Staubli VAL3: JPOINT.pjx

--- JPOINT.pjx ---
Parameters version=s7.6.1 stackSize=5000 millimeterUnit=true
Program file=computeFrame.pgx
Program file=delete.pgx
Program file=deleteItem.pgx
Program file=duplicate.pgx
Program file=find.pgx
Program file=get.pgx
Program file=getDistance.pgx
Program file=getFrame.pgx
Program file=getFrameId.pgx
Program file=getFunctionEdit.pgx
Program file=getFunctionSel.pgx
Program file=getFunctionView.pgx
Program file=getListItem.pgx
Program file=getPoint.pgx
Program file=getSize.pgx
Program file=getSizeItem.pgx
Program file=getTool.pgx
Program file=getTrajItem.pgx
Program file=getTrajType.pgx
Program file=goTo.pgx
Program file=HerePoint.pgx
Program file=insertItem.pgx
Program file=load.pgx
Program file=loadCycle.pgx
Program file=loadPage.pgx
Program file=makeTraj.pgx
Program file=moveTo.pgx
Program file=new.pgx
Program file=onEdit.pgx
Program file=onEditItem.pgx
Program file=onFunctionEdit.pgx
Program file=onFunctionSel.pgx
Program file=onFunctionView.pgx
Program file=onInsert.pgx
Program file=onProgEnd.pgx
Program file=onRun.pgx
Program file=onSave.pgx
Program file=onStart.pgx
Program file=onStop.pgx
Program file=setFrameId.pgx
Program file=setTool.pgx
Program file=setTrajItem.pgx
Data file=JPOINT.dtx
Library alias=saveData path=Disk://saveData/saveData.pjx
Library alias=page path=Disk://kernel/template/page/page.pjx
Library alias=use path=Disk://kernel/userPage/userPage.pjx
Library alias=language path=Disk://kernel/language/language.pjx
Library alias=tcp path=Disk://kernel/tool/tool.pjx
Library alias=cycleStatus path=Disk://cycleStatus/cycleStatus.pjx
Library alias=pt path=Disk://kernel/template/session/saveTraj/JPOINT/JPOINT.pjx
Library alias=home path=Disk://kernel/template/session/saveTraj/HOME/HOME.pjx
Type name=TrajectoryItem path=Disk://kernel/template/TrajectoryItem/TrajectoryItem.pjx
Type name=TrajJoint path=Disk://kernel/template/TrajJoint/TrajJoint.pjx
Type name=ActionItem path=Disk://kernel/template/ActionItem/ActionItem.pjx
Type name=InstrItem path=Disk://kernel/template/InstrItem/InstrItem.pjx
Type name=Trajectory path=Disk://kernel/template/Trajectory/Trajectory.pjx
Type name=TrajHome path=Disk://kernel/template/TrajHome/TrajHome.pjx
Type name=FrameItem path=Disk://kernel/template/FrameItem/FrameItem.pjx

--- JPOINT.dtx ---
public string sItems
string sPathTemplate = "Disk://kernel/template/JPOINT"
public bool bMoveType[3]
public bool bStepping
pointRx pToGo = {fatherId=world[0]}
pointRx pLastPoint = {fatherId=world[0]}
mdesc nom_speed = {accel=50, vel=50, decel=50, blend=off}
num nTcpAction
pointRx pPointTo = {fatherId=world[0]}
string sTrajType
string sMenu[8]
mdesc mMdesc = {accel=25, vel=25, decel=25, blend=off}
bool bToSave
InstrItem tcpInstr
  [0]
    string sType
    string sData
public Trajectory tTraj
  [0]
    TrajectoryItem tSuper
      [0]
        num distance
        num moveType
        num nTime
        num nStop
        num nTcpAction
        string comment
        bool toStop
        mdesc nom_speed = {tmax=300, rmax=9999, leave=30, reach=30}
        InstrItem iInstr[3]
          [0]
            string sType
            string sData
          [1]
            string sType
            string sData
          [2]
            string sType
            string sData
        num nMoveId
    string sID
    num nId
num nIndex
num nKey
TrajJoint jEditPoint
  [0]
    num nIndexTool
    TrajJointItem tData
      [0]
        jointRx jJoint
        TrajectoryItem tSuper
          [0]
            num distance
            num moveType
            num nTime
            num nStop
            num nTcpAction
            string comment
            bool toStop
            mdesc nom_speed = {tmax=9999, rmax=9999, leave=30, reach=30}
            InstrItem iInstr[3]
              [0]
                string sType
                string sData
              [1]
                string sType
                string sData
              [2]
                string sType
                string sData
            num nMoveId
    string sID
    num nIndexFrame
string sTrajCycle

--- delete.pgx ---
public program delete(string x_sName, num& x_nResult[])
  local string l_sItem
  local num l_nSize
begin
  //
  // delete the select trajectory
  //
  if isDefined(pt:tTraj[x_sName])
    // delete
    delete(pt:tTraj[x_sName])
    // save it
    bToSave=true
    x_nResult=0
  else
    x_nResult=-1
  endIf

end

--- deleteItem.pgx ---
public program deleteItem(num& x_nIndex)
  local num i
  local string l_sItem
begin
  // delete the selected item
  delete(jEditPoint.tData[x_nIndex])
end

--- duplicate.pgx ---
public program duplicate(string x_sCopy, string x_sPaste, num& x_nResult[])
  local num i
  local num l_nSize
  local string l_sItem
  local bool l_bFound
  local num l_nResult
  local string l_sString
  local num l_nX
  local num l_nY
begin
  // duplicate

  // look if the items exist
  if insert(pt:tTraj[x_sPaste])
    // link the point
    call pt:copy_it(x_sCopy,x_sPaste)
    call pt:link_it(x_sPaste)
    // save it
    bToSave=true
  endIf
end

--- find.pgx ---
public program find(string& x_sItem[], bool& x_bFound[])
begin
  // check if the item has been found
  x_bFound=isDefined(pt:tTraj[x_sItem])
end

--- getDistance.pgx ---
public program getDistance(tool x_tTool, num& x_nDistance[], bool x_bCycle, num x_nIndex)
  local num l_nDistance
  local point l_pPoint
  local num l_nValue
  local trsf l_trsfEmpty
begin
  // first point
  if x_nIndex==0
    x_nDistance=10
    return
  elseIf x_bCycle
    // an other one
    x_nDistance=distance(jointToPoint(x_tTool,world,pt:tTraj[sTrajCycle].tData[x_nIndex-1].jJoint),jointToPoint(x_tTool,world,pt:tTraj[sTrajCycle].tData[x_nIndex].jJoint))
  else
     x_nDistance=distance(jointToPoint(x_tTool,world,jEditPoint.tData[x_nIndex-1].jJoint),jointToPoint(x_tTool,world,jEditPoint.tData[x_nIndex].jJoint))
  endIf
end

--- getFunctionEdit.pgx ---
public program getFunctionEdit(string& x_sName[])
  local string l_sMessage
begin
  //
  // define your message for the
  // function KEY
  //
  // NOTE is an ARRAY[0..7]
  //
  // example:
  // x_sName[1]="DEMO"
  // active the F2 button
  //
  // here
  call language:message(l_sMessage,150)
  x_sName[0]=l_sMessage
  // ALIGN
  call language:message(l_sMessage,134)
  x_sName[1]=l_sMessage
  // Tool
  call language:message(l_sMessage,123)
  x_sName[2]=l_sMessage
end

--- getFunctionSel.pgx ---
public program getFunctionSel(string& x_sName[])
  local string l_sMessage
begin
  //
  // define your message for the
  // function KEY
  //
  // NOTE is an ARRAY[0..7]
  //
  // example:
  // x_sName[1]="DEMO"
  // active the F2 button
  //
end

--- getFunctionView.pgx ---
public program getFunctionView(string& x_sName[])
  local string l_sMessage
begin
  //
  // define your message for the
  // function KEY
  //
  // NOTE is an ARRAY[0..7]
  //
  // example:
  // x_sName[1]="DEMO"
  // active the F2 button
  //
  // here
  call language:message(l_sMessage,150)
  x_sName[0]=l_sMessage
  // ALIGN
  call language:message(l_sMessage,134)
  x_sName[1]=l_sMessage
end

--- getListItem.pgx ---
public program getListItem(string& x_sItem[], num x_nIndex)
  local trsf l_tTrsf
  local string l_sItem[6]
  local string l_sEvent
begin
  //
  //
  // define the item to show in the edit page Traj
  // customize an array and copy to x_sItem...
  //
  // see other traj as example
  l_sItem[0]=("Joint 1 > "+toString(".2",jEditPoint.tData[x_nIndex].jJoint.j1))
  l_sItem[1]=("Joint 2 > "+toString(".2",jEditPoint.tData[x_nIndex].jJoint.j2))
  l_sItem[2]=("Joint 3 > "+toString(".2",jEditPoint.tData[x_nIndex].jJoint.j3))
  l_sItem[3]=("Joint 4 > "+toString(".2",jEditPoint.tData[x_nIndex].jJoint.j4))
  l_sItem[4]=("Joint 5 > "+toString(".2",jEditPoint.tData[x_nIndex].jJoint.j5))
  l_sItem[5]=("Joint 6 > "+toString(".2",jEditPoint.tData[x_nIndex].jJoint.j6))
  call use:stringCopy(l_sItem,x_sItem)
end

--- getPoint.pgx ---
public program getPoint(point& x_pPoint[], bool x_bCycle, num x_nIndex)
  local string l_sItem
  local tool l_tTool
begin
  // take
  // check the point
  link(x_pPoint,world)
  if x_bCycle
    call tcp:getTool(l_tTool,pt:tTraj[sTrajCycle].nIndexTool)
    x_pPoint=jointToPoint(l_tTool,world,pt:tTraj[sTrajCycle].tData[x_nIndex].jJoint)
  else
    // give back the point
    call tcp:getTool(l_tTool,jEditPoint.nIndexTool)
    x_pPoint=jointToPoint(l_tTool,world,jEditPoint.tData[x_nIndex].jJoint)
  endIf
end

--- getSize.pgx ---
public program getSize(num& x_nSize[])
  local string l_sType
  local string l_sKey
  local num i
  local string l_sItem
  local string l_sPath
begin
  // give back the size to trajectory field
  x_nSize=size(pt:tTraj)
end

--- getSizeItem.pgx ---
public program getSizeItem(bool x_bCycle, num& x_nSize)
  local string l_sType
  local string l_sKey
  local num i
begin
  //
  // get the size of the collection
  //
  if x_bCycle
    x_nSize=size(pt:tTraj[sTrajCycle].tData)
  else
    x_nSize=size(jEditPoint.tData)
  endIf
end

--- getTrajItem.pgx ---
public program getTrajItem(TrajectoryItem& x_tTraj[], num x_nIndex)
begin
  //
  // get all the FIELD
  //
  x_tTraj=jEditPoint.tData[x_nIndex].tSuper
end

--- goTo.pgx ---
public program goTo(tool x_tTool, mdesc x_mDesc, num x_nMoveType, bool& x_bUnreached[], num x_nIndex)
  local point l_pTrsf
  local bool l_bInside
  local tool l_tTool
  local point l_pHere
  local string l_sMessage
  local num l_nSize
  local num i
begin
  // the maximum size
  if isInRange(jEditPoint.tData[x_nIndex].jJoint)
    // go to the select Joint
    movej(jEditPoint.tData[x_nIndex].jJoint,x_tTool,x_mDesc)
  else
    x_bUnreached=true
  endIf
end

--- HerePoint.pgx ---
public program HerePoint(num x_nIndex)
  local tool l_tTool
  local point l_pHere
  local frame l_fFrame
  local num i
  local num l_nIndex
begin
  //
  // take the point
  //
  jEditPoint.tData[x_nIndex].jJoint=herej()
  resetMotion()
end

--- insertItem.pgx ---
public program insertItem(num x_nIndexCopy, num x_nIndexPaste)
  local num l_nLastType
  local point l_pPoint
  local num l_nType
  local joint l_jJoint
begin
  //
  // use to add more elements from the typical one
  //
  // insert all the field
  //
  // JOINT
  l_jJoint=jEditPoint.tData[x_nIndexCopy].jJoint
  insert(jEditPoint.tData[x_nIndexPaste])
  jEditPoint.tData[x_nIndexPaste].jJoint=l_jJoint

end

--- load.pgx ---
public program load(string x_sItem, num& x_nResult)
  local string l_sType
  local string l_sMessage
begin
  // load the select trajectory..already loaded
  call getTrajType(l_sType)
  if find(pt:libPath(),saveData:sPathTraj)==-1
    pt:libLoad(saveData:sPathTraj+l_sType)
    delay(0)
    if saveData:bDebug
      ? "loading JPOINT..."+saveData:sPathTraj+l_sType
    endIf
  endIf
  // use the type...
  if isDefined(pt:tTraj[x_sItem])
    // use the type...
    jEditPoint=pt:tTraj[x_sItem]
    jEditPoint.sID=x_sItem
    x_nResult=0
  elseIf x_sItem!="" and find(x_sItem,"@")==-1
    // not FOUND
    call language:message(l_sMessage,-7)
    x_nResult=-1
    popUpMsg(l_sMessage+x_sItem)
    jEditPoint.sID=""
  elseIf x_sItem==""
    // reload all the template
    x_nResult=home:libLoad(saveData:sPathTraj+"HOME")
    if saveData:bDebug
      ? "loading JPOINT HOME..."+saveData:sPathTraj+"HOME"
    endIf
  endIf
end

--- loadCycle.pgx ---
public program loadCycle(string x_sItem, num& x_nResult[])
  local string l_sType
  local string l_sMessage
begin
  // load the select trajectory..already loaded
  call getTrajType(l_sType)
  if find(pt:libPath(),saveData:sPathTraj)==-1
    pt:libLoad(saveData:sPathTraj+l_sType)
    delay(0)
    if saveData:bDebug
      ? "loading JPOINT..."+saveData:sPathTraj+l_sType
    endIf
  endIf
  if isDefined(pt:tTraj[x_sItem])
    // use the type...
    sTrajCycle=x_sItem
  else
    // not FOUND
    call language:message(l_sMessage,-7)
    x_nResult=-1
    cycleStatus:bToStop=true
    popUpMsg(l_sMessage+x_sItem)
  endIf
end

--- loadPage.pgx ---
program loadPage(string x_sPage, string& x_sItems[])
// load the next page
  local num i
begin
  // look if the page libload is correct
  i=page:libLoad(x_sPage)
    delay(0)
  logMsg("KERNEL:PAGE LIBLOAD "+x_sPage+" result "+toString("",i))
  if i!=0
    popUpMsg("Loading page "+x_sPage+" error CODE "+toString("",i))
  else
    page:sItems=x_sItems
    call page:main()
  endIf
end

--- makeTraj.pgx ---
public program makeTraj(string& x_sItem[])
  local num i
  local num l_nSize
  local tool l_tTool
  local bool l_bUnreached
  local point l_pPoint[2]
  local num l_nMoveId
  local bool l_bOk
  local ActionItem l_aAction
  local num j
  local TrajectoryItem l_tTraj
  local num l_nDistance
  local joint l_jJoint
  local Trajectory l_tTrajectory
begin
  //
  // inizialize the system
  //
  // take the TOOL
  call tcp:getTool(l_tTool,pt:tTraj[sTrajCycle].nIndexTool)
  //
  // for all of my traj cycleJoint move the robot
  //
  // the maximum size
  call getSizeItem(true,l_nSize)
  //
  // for all of my traj cyclePoints move the robot
  //
  resize(tTraj.tSuper,1,size(pt:tTraj[sTrajCycle].tData))
  for i=0 to (l_nSize-1)
    tTraj.tSuper[i]=pt:tTraj[sTrajCycle].tData[i].tSuper
  endFor
  tTraj.sID="JPOINT "+pt:tTraj[sTrajCycle].sID
  call cycleStatus:addTraj(tTraj)
  for i=0 to (l_nSize-1)
    //
    // get the point info
    //
    l_tTraj=pt:tTraj[sTrajCycle].tData[i].tSuper
    //
    // get the distance in percentage
    //
    call getDistance(l_tTool,l_nDistance,true,i)
    //
    // give to the traj library the percentage distance
    //
    if l_tTraj.toStop
      l_tTraj.nom_speed.blend=off
    endIf
    //
    // put the move in the stack
    //
    l_jJoint=pt:tTraj[sTrajCycle].tData[i].jJoint
    call moveTo(l_tTool,l_tTraj.nom_speed,l_tTraj.moveType,l_bUnreached,l_jJoint,l_nMoveId)
    // set the data
    l_aAction.nDistance=l_nDistance
    l_aAction.nPointId=i
    l_aAction.nMoveId=l_nMoveId
    l_aAction.sIdTraj="JPOINT "+pt:tTraj[sTrajCycle].sID
    call cycleStatus:putInstr_Traj(l_aAction,l_tTraj,pt:tTraj[sTrajCycle].nIndexTool,l_nSize)
    // there is a waitEndMove
    if l_tTraj.toStop
      waitEndMove()
      delay(l_tTraj.nStop)
      // wait all the action has been done
      wait(cycleStatus:bActionRunning==false)
    endIf
  endFor
end

--- moveTo.pgx ---
public program moveTo(tool x_tTool, mdesc x_mDesc, num x_nMoveType, bool& x_bUnreached[], joint& x_jJoint[], num& x_nMoveId)
begin
  //
  // use the percentage speed
  //
  x_mDesc.vel=saveData:nSpeed/100*x_mDesc.vel
  x_nMoveId=movej(x_jJoint,x_tTool,x_mDesc)
end

--- onEdit.pgx ---
public program onEdit(string& x_sItem[])
  local string l_sPath
  local num i
  local string l_sItem
  local num l_nSize
  local TrajectoryItem l_tTraj
  local num l_nResult
  local string l_sPoint
begin
  // DEFINE YOUR ITEM
  call getTrajType(saveData:sTrajTypeUsing)
  // load the trajectory
  call load(x_sItem,l_nResult)
  if find(x_sItem,"@")==-1
    // load the page viewTraj
    l_sPath="Disk://trajectory/page_viewTraj"
    // give back the path
    x_sItem[1]=x_sItem
    x_sItem=l_sPath
  endIf
end

--- onEditItem.pgx ---
public program onEditItem(string& x_sEvent[], num x_nIndex, num x_nIndexItem)
  local joint l_jJoint
  local num i
  local string l_sEmpty
  local string l_sMessage
begin
  // edit the custom element that was add in the list
  l_jJoint=jEditPoint.tData[x_nIndexItem].jJoint
  call use:findPos(x_sEvent,">",i)
  i=i+1
  // clean the line
  call use:listcursor(use:nView,false)
  l_sEmpty=""
  switch x_nIndex
    case 0
      //  j1-value
      if cycleStatus:bCycle
        // set a limit +- 5
        call use:changeValue(l_jJoint.j1,l_jJoint.j1-5,l_jJoint.j1+5,i+40-use:nBottomX,use:nView+1,l_sEmpty)
      else
        call use:changeValue(l_jJoint.j1,0,0,i+40-use:nBottomX,use:nView+1,l_sEmpty)
      endIf
    break
    case 1
      //  j2-value
      if cycleStatus:bCycle
        // set a limit +- 5
        call use:changeValue(l_jJoint.j2,l_jJoint.j2-5,l_jJoint.j2+5,i+40-use:nBottomX,use:nView+1,l_sEmpty)
      else
        call use:changeValue(l_jJoint.j2,0,0,i+40-use:nBottomX,use:nView+1,l_sEmpty)
      endIf
    break
    case 2
      //  j3-value
      if cycleStatus:bCycle
        // set a limit +- 5
        call use:changeValue(l_jJoint.j3,l_jJoint.j3-5,l_jJoint.j3+5,i+40-use:nBottomX,use:nView+1,l_sEmpty)
      else
        call use:changeValue(l_jJoint.j3,0,0,i+40-use:nBottomX,use:nView+1,l_sEmpty)
      endIf
    break
    case 3
      //  j4-value
      if cycleStatus:bCycle
        // set a limit +- 5
        call use:changeValue(l_jJoint.j4,l_jJoint.j4-5,l_jJoint.j4+5,i+40-use:nBottomX,use:nView+1,l_sEmpty)
      else
        call use:changeValue(l_jJoint.j4,0,0,i+40-use:nBottomX,use:nView+1,l_sEmpty)
      endIf
    break
    case 4
      //  j5-value
      if cycleStatus:bCycle
        // set a limit +- 5
        call use:changeValue(l_jJoint.j5,l_jJoint.j5-5,l_jJoint.j5+5,i+40-use:nBottomX,use:nView+1,l_sEmpty)
      else
        call use:changeValue(l_jJoint.j5,0,0,i+40-use:nBottomX,use:nView+1,l_sEmpty)
      endIf
    break
    case 5
      //  j6-value
      if cycleStatus:bCycle
        // set a limit +- 5
        call use:changeValue(l_jJoint.j6,l_jJoint.j6-5,l_jJoint.j6+5,i+40-use:nBottomX,use:nView+1,l_sEmpty)
      else
        call use:changeValue(l_jJoint.j6,0,0,i+40-use:nBottomX,use:nView+1,l_sEmpty)
      endIf
    break
  endSwitch
  //
  if isInRange(l_jJoint)
    jEditPoint.tData[x_nIndexItem].jJoint=l_jJoint
  else
    // error using the trsf
    call language:message(l_sMessage,-5)
    popUpMsg(l_sMessage)
  endIf
  // wait no key
  call use:nullKey(nKey)
end

--- onFunctionEdit.pgx ---
public program onFunctionEdit(num x_nIndex, string x_sEvent, num x_nFunctionKey)
  local string l_sMessage
  local string l_sButton[2]
  local bool l_bOk
  local string l_sPage
  local string l_sItem
  local tool l_tTool
  local point l_pAlign
  local bool l_bYes
  local string l_sMessage2
begin
  //
  // do on Key action
  //
  // x_nIndex = actual index item
  // x_sEvent = actual event item
  //
  switch x_nFunctionKey
    // F1 button
    case 271
      // HERE JOINT
      if !cycleStatus:bCycle
        call language:message(l_sMessage,160)
        call language:getYesNo(l_sButton)
        // ask the yes_no question
        call use:yes_no(l_sMessage,l_sButton,l_bYes)
        if l_bYes
          call HerePoint(x_nIndex)
        endIf
      endIf
    break
    case 272
      // ALIGN
      if !cycleStatus:bCycle
        resetMotion()
        // tool
        call tcp:getTool(l_tTool,jEditPoint.nIndexTool)
        l_pAlign=here(l_tTool,world)
        l_pAlign.trsf=align(l_pAlign.trsf,saveData:fFrameItem[saveData:nFrameActive].fFrame.trsf)
        call language:message(l_sMessage,203)
        call language:message(l_sMessage2,134)
        l_sMessage=l_sMessage+" "+l_sMessage2+"..."
        call use:timerDialog(l_sMessage,0)
        movej(l_pAlign,l_tTool,mMdesc)
        watch(isEmpty() or isKeyPressed(255),3)
        if !isEmpty()
          resetMotion()
        endIf
        delay(2)
      endIf
    break
    // F3 button
    case 273
      // Select the gun
      l_sPage="Disk://kernel/page/tool"
      call loadPage(l_sPage,l_sItem)
      // set the tool
      jEditPoint.nIndexTool=saveData:nIndexTool
    break
    // F4 button
    case 274
    break
    // F5 button
    case 275
    break
    // F6 button
    case 276
    break
    // F7 button
    case 277
    break
    // F8 button
    case 278
      // save it
    break
  endSwitch
end

--- onFunctionSel.pgx ---
public program onFunctionSel(num x_nIndex, string& x_sEvent, num x_nFunctionKey)
  local num l_nX
  local num l_nY
  local string l_sString
  local string l_sName
begin
  //
  // do on Key action
  //
  // x_nIndex = actual index item
  // x_sEvent = actual event item
  //
  l_nX=40-use:nBottomX-1
  l_nY=use:nBottomY+1
  switch x_nFunctionKey
    // F1 button
    case 271
    break
    // F2 button
    case 272
    break
    // F3 button
    case 273
    break
    // F4 button
    case 274
    break
    // F5 button
    case 275
    break
    // F6 button
    case 276
    break
    // F7 button
    case 277
    break
    // F8 button
    case 278
      //      call language:message(l_sString,21)
      //      call use:type(l_nX,l_nY,l_sString)
      //      // read the new trajectory
      //      call use:read(l_nX+len(l_sString),l_nY,l_sName,10,false)
      //      if !use:bUseEscape
      //        // look if the items exist
      //        if insert(pt:tTraj[l_sName])
      //          call pt:link_it(l_sName)
      //          pt:tTraj[l_sName].nIndexTool=saveData:nIndexTool
      //          // save it
      //          bToSave=true
      //          // export
      //          x_sEvent=l_sName
      //        else
      //          call language:message(l_sString,-2)
      //          popUpMsg(l_sString)
      //        endIf
      //      endIf
    break
  endSwitch
end

--- onFunctionView.pgx ---
public program onFunctionView(num x_nIndex, string x_sEvent, num x_nFunctionKey)
  local string l_sMessage
  local string l_sButton[2]
  local bool l_bYes
  local tool l_tTool
  local point l_pAlign
  local string l_sMessage2
  local joint l_jJoint
  local num l_nIndexFrame
  local frame l_fFrame
begin
  //
  // do on Key action
  //
  // x_nIndex = actual index item
  // x_sEvent = actual event item
  //
  switch x_nFunctionKey
    // F1 button
    case 271
      // HERE JOINT
      if !cycleStatus:bCycle
        call language:message(l_sMessage,160)
        call language:getYesNo(l_sButton)
        // ask the yes_no question
        call use:yes_no(l_sMessage,l_sButton,l_bYes)
        if l_bYes
          call HerePoint(x_nIndex)
        endIf
      endIf
    break
    // F2 button
    case 272
      // ALIGN
      if !cycleStatus:bCycle and !cycleStatus:bSimulation
        resetMotion()
        call getFrameId(l_nIndexFrame)
        l_fFrame=saveData:fFrameItem[l_nIndexFrame].fFrame
        // tool
        call tcp:getTool(l_tTool,jEditPoint.nIndexTool)
        l_pAlign=here(l_tTool,l_fFrame)
        l_pAlign.trsf=align(l_pAlign.trsf,l_fFrame.trsf)
        // check the align
        if pointToJoint(l_tTool,herej(),l_pAlign,l_jJoint)
          call language:message(l_sMessage,203)
          call language:message(l_sMessage2,134)
          l_sMessage=l_sMessage+" "+l_sMessage2+"..."
          call use:timerDialog(l_sMessage,0)
          movel(l_pAlign,l_tTool,mMdesc)
          watch(isEmpty() or isKeyPressed(255),3)
          if !isEmpty()
            resetMotion()
          endIf
          delay(2)
        endIf
      endIf
    break
    // F3 button
    case 273
    break
    // F4 button
    case 274
    break
    // F5 button
    case 275
    break
    // F6 button
    case 276
    break
    // F7 button
    case 277
    break
    // F8 button
    case 278
    break
  endSwitch
end

--- onInsert.pgx ---
public program onInsert(string& x_sItem[])
  local string l_sEvent
  local num l_nKey
  local num l_nIndex
  local num l_nSize
  local num i
  local string l_sMessage
  local bool l_bFound
  local string l_sType
  local bool l_bUseFilter
  local string l_sPaste
  local num l_nResult
  local num l_nX
  local num l_nY
  local string l_sName
begin
  // get the type
  call getTrajType(x_sItem)
  saveData:sTrajTypeUsing=x_sItem
  cls()
  // is a filter using ??
  if saveData:sTrajFilter!=""
    l_bUseFilter=true
    call language:message(l_sMessage,64)
    call use:type(0,1,l_sMessage+">ON")
  else
    // clean
    call use:typeLen(0,1," ",use:nBottomX)
  endIf
  //
  // CREATE THE LIST
  //
  // define your list size for default
  call use:setSizeList(19,0,19,11)
  call use:setView(false)
  call use:listcreate(x_sItem)
  // take the coordinate....
  l_nX=40-use:nBottomX-1
  l_nY=use:nBottomY+1
  // show the message
  call language:message(l_sMessage,61)
  call use:stringToArray(l_sMessage,sMenu)
  // insert the HOME POINT
  call language:message(l_sMessage,190)
  sMenu[0]="HOME "+l_sMessage
  call use:setMenu(sMenu,true,3)
  // Build the list
  call getSize(l_nSize)
  for i=0 to l_nSize-1
    call get(l_sEvent,i)
    if l_sEvent!=""
      //
      // use the filter ?
      //
      // check if the bProcessList filter is active
      //
      l_bFound=true
      if saveData:sTrajFilter!=""
        l_bFound=find(l_sEvent,saveData:sTrajFilter)!=-1
      endIf
      // add
      if l_bFound
        call use:listadd(l_sEvent)
      endIf
    endIf
  endFor
  call use:listupdate(0)
  do
    // get the item
    l_nKey=get()
    call use:listevent(l_nKey,l_nIndex,l_sEvent)
    if l_nKey==271 and l_bUseFilter
      // Build the list
      call getSize(l_nSize)
      // empty and rebuild
      call use:listempty()
      for i=0 to l_nSize-1
        call get(l_sEvent,i)
        if l_sEvent!=""
          call use:listadd(l_sEvent)
        endIf
      endFor
      // clean
      call use:typeLen(0,1," ",use:nBottomX)
      call use:typeMenu(1," ")
      l_bUseFilter=false
      call use:listupdate(0)
    endIf
    //
  until l_nKey==270 or l_nKey==255 or l_nKey==278 or l_nKey==276 or l_nKey==271
  //
  switch l_nKey
    case 270
      // save the name
      l_sName=l_sEvent
    break
    case 271
      // insert the home Point
      l_sName="@HOME"
    break
    case 276
      // duplicate
      // ask for the new
      call language:message(l_sMessage,21)
      call use:type(l_nX,l_nY,l_sMessage)
      l_sName=l_sEvent
      // read the new trajectory
      call use:read(l_nX+len(l_sMessage),l_nY,l_sName,10,false)
      if !use:bUseEscape
        call duplicate(l_sEvent,l_sName,l_nResult)
      endIf
    break
    case 278
      call language:message(l_sMessage,21)
      call use:type(l_nX,l_nY,l_sMessage)
      // read the new trajectory
      call use:read(l_nX+len(l_sMessage),l_nY,l_sName,10,false)
      if !use:bUseEscape
        // look if the items exist
        call new(l_sName,l_nResult)
        if l_nResult==-1
          call language:message(l_sMessage,-2)
          popUpMsg(l_sMessage)
        endIf
      endIf
    break
  endSwitch
  if l_nKey!=255
    x_sItem=l_sName
  else
    x_sItem=""
  endIf
  call use:nullKey(l_nKey)
end

--- onRun.pgx ---
public program onRun(string& x_sItem[])
  local string l_sEmpty
  local num l_nResult
  local num l_nIndex
  local mdesc l_mDesc
  local bool l_bUnreached
  local num l_nMoveId
  local string l_sComment
  local Trajectory l_tTraj
  local joint l_jJoint
begin
  if find(x_sItem,"@HOME")!=-1
    //load the home home
    l_nResult=home:libLoad(saveData:sPathTraj+"HOME")
    delay(0)
    l_nIndex=size(home:tTraj["home"].tData)-1
    l_mDesc=home:tTraj["home"].tData[l_nIndex].tSuper.nom_speed
    l_jJoint=home:tTraj["home"].tData[l_nIndex].jJoint
    // execute the movement
    call moveTo(flange,l_mDesc,0,l_bUnreached,l_jJoint,l_nMoveId)
    // show the comments
    l_tTraj.tSuper=home:tTraj["home"].tData[l_nIndex].tSuper
    l_tTraj.sID="JPOINT @HOME"
    call cycleStatus:addTraj(l_tTraj)
    wait(getMoveId()>=l_nMoveId-0.1 or isEmpty())
  else
    // execute check if need to reload
    call loadCycle(x_sItem,l_nResult)
    if l_nResult==0
      // execute
      call makeTraj(x_sItem)
    else
      popUpMsg("JOINT NOT DEFINE !!!")
      cycleStatus:bToStop=false
    endIf
  endIf
end

--- onSave.pgx ---
public program onSave(string& x_sItem[])
  local num i
  local num l_nSize
begin
  //if bToSave
  // update
  if isDefined(pt:tTraj[jEditPoint.sID])
    pt:tTraj[jEditPoint.sID]=jEditPoint
  endIf
  // saveIt
  pt:libSave()
  bToSave=false
  //endIf
end

--- onStart.pgx ---
public program onStart(string& x_sItem[])
  local num i
  local string l_sType
begin
end

--- onStop.pgx ---
public program onStop(string& x_sItem[])
begin
  // stop it
  if x_sItem=="kill"
    pt:libLoad("Disk://kernel/template/session/saveTraj/JPOINT")
  endIf
end

--- setFrameId.pgx ---
public program setFrameId(num x_nIndex)
begin
  // set the Frame
  jEditPoint.nIndexFrame=x_nIndex
end

--- setTool.pgx ---
public program setTool(num x_nIndexTool)
begin
  // set the TOOL
  jEditPoint.nIndexTool=x_nIndexTool
end
